// TIA Portal V20 export
FUNCTION_BLOCK "CallInterfaceSignalsConv"   // FB213, LAD
// stored: MemoryReserve 100, SetENOAutomatically false
   VAR_INPUT
      InterfaceTestMode : Bool;
   END_VAR
   VAR_OUTPUT
      signals_I2S : "typeInspectionToStack";
      signals_S2I : "typeStackToInspection";
   END_VAR
   VAR_IN_OUT
      Comm_I2S : Array[0..95] of Bool;
      Comm_S2I : Array[0..95] of Bool;
      InterfaceTestButton : "LER_SignalsInput";
   END_VAR
   VAR
      statWordBuffer_I2S : Array[0..5] of Word;
      statWordBuffer_S2I : Array[0..5] of Word;
   END_VAR
   VAR_TEMP
      tempDeleteData : "LER_SignalsInput";
   END_VAR
   VAR CONSTANT
      TRUE : Bool := TRUE;
   END_VAR
   VAR_TEMP   // added for the SCL form of the ladder/FBD networks
      _w1 : Bool;
      _w2 : Bool;
      _w3 : Bool;
      _w4 : Bool;
   END_VAR
BEGIN

REGION Network 1: CommI2S -> signalsI2S
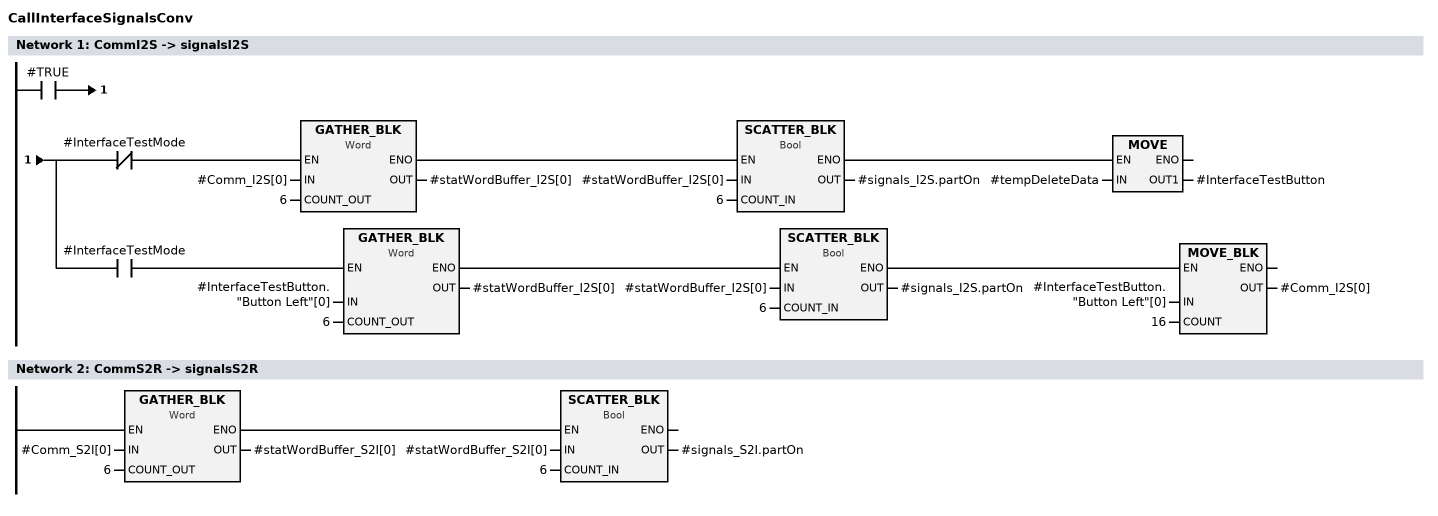
   GATHER_BLK(EN := #TRUE AND NOT #InterfaceTestMode,
              IN := #Comm_I2S[0],
              COUNT_OUT := 6,
              OUT => #statWordBuffer_I2S[0],
              ENO => #_w1);
   SCATTER_BLK(EN := #_w1, IN := #statWordBuffer_I2S[0], COUNT_IN := 6, OUT => #signals_I2S.partOn, ENO => #_w2);
   IF #_w2 THEN #InterfaceTestButton := #tempDeleteData; END_IF;
   GATHER_BLK(EN := #TRUE AND #InterfaceTestMode,
              IN := #InterfaceTestButton."Button Left"[0],
              COUNT_OUT := 6,
              OUT => #statWordBuffer_I2S[0],
              ENO => #_w3);
   SCATTER_BLK(EN := #_w3, IN := #statWordBuffer_I2S[0], COUNT_IN := 6, OUT => #signals_I2S.partOn, ENO => #_w4);
   IF #_w4 THEN
       MOVE_BLK(IN := #InterfaceTestButton."Button Left"[0], COUNT := 16, OUT => #Comm_I2S[0]);
   END_IF;
END_REGION

REGION Network 2: CommS2R -> signalsS2R
   RUNG wire#powerrail
      { S7_Templates := "[dest_type := Word, src_type := Bool, count_type := UInt]" } GATHER_BLK(IN := #Comm_S2I[0], COUNT_OUT := 6, OUT => #statWordBuffer_S2I[0])
      { S7_Templates := "[dest_type := Bool, src_type := Word, count_type := UInt]" } SCATTER_BLK(IN := #statWordBuffer_S2I[0], COUNT_IN := 6, OUT => #signals_S2I.partOn)
   END_RUNG
   // the same network as SCL:
   GATHER_BLK(IN := #Comm_S2I[0], COUNT_OUT := 6, OUT => #statWordBuffer_S2I[0], ENO => #_w1);
   IF #_w1 THEN SCATTER_BLK(IN := #statWordBuffer_S2I[0], COUNT_IN := 6, OUT => #signals_S2I.partOn); END_IF;
END_REGION
END_FUNCTION_BLOCK
